TYPE "UDT_ZC_RECETA_BATCH"
VERSION : 0.1
   STRUCT
      Id : Int;
      Nombre : String;
      Etapa { S7_SetPoint := 'False'} : Array[0..4] of "UDT_ZC_RECETA_BATCH_ETAPA";
   END_STRUCT;

END_TYPE

